Fanuc KAREL source: kt00330.KL

-- PROVISIONAL review KL for V770-1; original PC SHA256 94ae38df9015df1aefff2e70cacaad7423666b80d77e96d7a1668266e035f1ea
-- Incomplete behavior may be omitted. Consult companion uncertainty JSON. Do not deploy.
PROGRAM KT00330
%NOLOCKGROUP
VAR
  I1 : INTEGER
  R2 : REAL
  OUT : BOOLEAN
BEGIN
  -- UNRESOLVED_PC offsets 5-16; opcodes 2E,23
  -- UNRESOLVED_PC offsets 21-32; opcodes 2E,23
  -- UNRESOLVED_PC offsets 37-59; opcodes 21,21,29,64,29,6F,23
  -- UNRESOLVED_PC offsets 64-68; opcodes 7F
END KT00330
